(* PLC project flow_compute, Dassault Systèmes ControlBuild 2024x *)
(* stored: creationDateTime 2023-10-03T11:13:02-01:00 *)

(* This module computes the flow in litre / min. It should be set at the inlet of the circuit or at the outlet of a tank. *)
FUNCTION_BLOCK equipment_library.flow_compute
  VAR_INPUT
    inputFlow : REAL := 0.0;
  END_VAR
  VAR_OUTPUT
    outputFlow : REAL := 0.0;
  END_VAR
  VAR
    unit : REAL := 0.0;
  END_VAR
  VAR CONSTANT
    flowMax : REAL := 200.0;
    flowPerHour : BOOL := true;
    flowPerMinute : BOOL := false;
  END_VAR


ACTION C_source_code:
/* -----------------------------------------------------------------	*/
/* Type : Model of Operative Behaviour					*/
/* Catégorie :   batch							*/
/* Author : Dassault Systemes						*/
/* Update date : June 2018							*/
/* -----------------------------------------------------------------	*/
/* This module computes the flow in litre / min.			*/
/* It should be set at the inlet of the circuit or at the outlet of	*/
/* a tank.									*/
/* ----------------------------------------------------------------	*/

if (flowPerHour) unit = 3600.0;
else if (flowPerMinute) unit = 60.0;
	else unit = 1.0;

outputFlow = (flowMax * CLOCK_PERIOD / 1000000) / unit;

if (inputFlow < outputFlow)
	outputFlow = inputFlow;
END_ACTION
END_FUNCTION_BLOCK
